fbMR1K4_Coating_States.stCoating2.stPMPS.sPmpsState := 'MR1K4:SOMS-B4C';
fbMR1K4_Coating_States.stCoating2.nEncoderCount := 5000141;

fbMR2K4_Coating_States.stCoating1.stPMPS.sPmpsState := 'MR2K4:KBO-SILICON';
fbMR2K4_Coating_States.stCoating1.nEncoderCount := 8701960;

fbMR2K4_Coating_States.stCoating2.stPMPS.sPmpsState := 'MR2K4:KBO-B4C';
fbMR2K4_Coating_States.stCoating2.nEncoderCount := 6636177;

fbMR3K4_Coating_States.stCoating1.stPMPS.sPmpsState := 'MR3K4:KBO-SILICON';
fbMR3K4_Coating_States.stCoating1.nEncoderCount := 4719890;

fbMR3K4_Coating_States.stCoating2.stPMPS.sPmpsState := 'MR3K4:KBO-B4C';
fbMR3K4_Coating_States.stCoating2.nEncoderCount := 8220029;

fbMR1K4_Coating_States(
    bEnable := TRUE,
    stMotionStage:=Main.M1,
    sCoating1Name:='Si',
    sCoating2Name:='B4C',
    fbArbiter:=GVL_PMPS.g_fbArbiter1,
    fbFFHWO:=GVL_PMPS.g_FastFaultOutput1,
    sPmpsDeviceName:='MR1K4:SOMS',
    sTransitionKey:= 'MR1K4:SOMS-TRANSITION');

// MR2K4 Coating States with PMPS
fbMR2K4_Coating_States(
    bEnable := TRUE,
    stMotionStage:=Main.M8,
    sCoating1Name:='Si',
    sCoating2Name:='B4C',
    fbArbiter:=GVL_PMPS.g_fbArbiter2,
    fbFFHWO:=GVL_PMPS.g_FastFaultOutput2,
    sPmpsDeviceName:='MR2K4:KBO',
    sTransitionKey:= 'MR2K4:KBO-TRANSITION'
);

// MR3K4 Coating States with PMPS
fbMR3K4_Coating_States(
    bEnable := TRUE,
    stMotionStage:=Main.M12,
    bVerticalCoating:=FALSE,
    sCoating1Name:='Si',
    sCoating2Name:='B4C',
    fbArbiter:=GVL_PMPS.g_fbArbiter2,
    fbFFHWO:=GVL_PMPS.g_FastFaultOutput2,
    sPmpsDeviceName:='MR3K4:KBO',
    sTransitionKey:= 'MR3K4:KBO-TRANSITION'
);

fbMR4K4XSetup(stPositionState:= fbMR4K4Default, bSetDefault :=TRUE);
fbMR4K4XSetup(stPositionState:=aMR4K4CoatingStatesX[ENUM_Si_B4C_Coating_States_1D.B4C],
    sName:='B4C',
    sPmpsState:='MR4K4:KBO-B4C',
    fDelta := 4.187,
    nEncoderCount:= 6727471
);
fbMR4K4XSetup(stPositionState:=aMR4K4CoatingStatesX[ENUM_Si_B4C_Coating_States_1D.Si],
    sName:='Si',
    sPmpsState:='MR4K4:KBO-SILICON',
    fDelta := 3.65,
    nEncoderCount:= 4322111
);
fbMR4K4_Coating_States(
    stMotionStage:=Main.M17,
    astPositionState:= aMR4K4CoatingStatesX,
    eEnumSet:= eMR4K4StateSet,
    eEnumGet:= eMR4K4StateGet,
    fbArbiter:=GVL_PMPS.g_fbArbiter2,
    fbFFHWO:=GVL_PMPS.g_FastFaultOutput3,
    bEnableMotion:=TRUE,
    bEnableBeamParams:=TRUE,
    sDeviceName:='MR4K4:KBO',
    sTransitionKey:= 'MR4K4:KBO-TRANSITION');

fbMR5K4YSetup(stPositionState:= fbMR5K4Default, bSetDefault :=TRUE);
fbMR5K4YSetup(stPositionState:=aMR5K4CoatingStatesY[ENUM_Si_B4C_Coating_States_1D.B4C],
    sName:='B4C',
    sPmpsState:='MR5K4:KBO-B4C',
    fDelta := 7.85,
    nEncoderCount:= 6785425
);
fbMR5K4YSetup(stPositionState:=aMR5K4CoatingStatesY[ENUM_Si_B4C_Coating_States_1D.Si],
    sName:='Si',
    sPmpsState:='MR5K4:KBO-SILICON',
    fDelta := 3.55,
    nEncoderCount:= 4265000
);
fbMR5K4_Coating_States(
    stMotionStage:=Main.M22,
    astPositionState:= aMR5K4CoatingStatesY,
    eEnumSet:= eMR5K4StateSet,
    eEnumGet:= eMR5K4StateGet,
    fbArbiter:=GVL_PMPS.g_fbArbiter2,
    fbFFHWO:=GVL_PMPS.g_FastFaultOutput3,
    bEnableMotion:=TRUE,
    bEnableBeamParams:=TRUE,
    sDeviceName:='MR5K4:KBO',
    sTransitionKey:= 'MR5K4:KBO-TRANSITION');

END_PROGRAM

// ---- POUs/PRG_PMPS.TcPOU
PROGRAM PRG_PMPS
VAR
    fb_vetoArbiter : FB_VetoArbiter;

    fbArbiterIO : FB_SubSysToArbiter_IO;

    ffFFO2ToFFO1 : FB_FastFault := (
        i_xAutoReset := TRUE,
        i_DevName := 'PMPS FFO2',
        i_Desc := 'Subordinate fast fault group, will clear on its own otherwise something is misconfigured in the diagnostic',
        i_TypeCode := 16#D);
//adding FFO3 for dream mirror so that we can veto dream mirror by ST4K4
   ffFFO3ToFFO1 : FB_FastFault := (
        i_xAutoReset := TRUE,
        i_DevName := 'PMPS FFO3',
        i_Desc := 'Subordinate fast fault group, will clear on its own otherwise something is misconfigured in the diagnostic',
        i_TypeCode := 16#D);

 //fbOutputStates : FB_StateParams;

    bMR1K1_IN : BOOL;
    bST3K4_IN : BOOL;
    bMR1K3_IN : BOOL;
    bST1K0_IN : BOOL;
    bST4K4_IN : BOOL;
END_VAR

MOTION_GVL.fbStandardPMPSDB(
    io_fbFFHWO:= GVL_PMPS.g_FastFaultOutput1,
    bEnable:=TRUE,
    sPLCName:='plc-tmo-optics'
);

P_StripeProtections();

bMR1K1_IN := PMPS.PMPS_GVL.stCurrentBeamParameters.aVetoDevices[PMPS.K_Stopper.MR1K1_IN]
            AND NOT PMPS.PMPS_GVL.stCurrentBeamParameters.aVetoDevices[PMPS.K_Stopper.MR1K1_OUT];

bST3K4_IN := PMPS.PMPS_GVL.stCurrentBeamParameters.aVetoDevices[PMPS.K_Stopper.ST3K4];
bST1K0_IN := PMPS.PMPS_GVL.stCurrentBeamParameters.aVetoDevices[PMPS.K_Stopper.ST1K0];

bMR1K3_IN := PMPS.PMPS_GVL.stCurrentBeamParameters.aVetodevices[PMPS.K_Stopper.MR1K3_IN]
    AND NOT PMPS.PMPS_GVL.stCurrentBeamParameters.aVetoDevices[PMPS.K_Stopper.MR1K3_OUT];

bST4K4_IN := PMPS.PMPS_GVL.stCurrentBeamParameters.aVetoDevices[PMPS.K_Stopper.ST4K4];

fbArbiterIO(i_bVeto:= bMR1K1_IN OR bMR1K3_IN, Arbiter := GVL_PMPS.g_fbArbiter1, fbFFHWO := GVL_PMPS.g_FastFaultOutput1);

ffFFO2ToFFO1(i_xOK := GVL_PMPS.g_FastFaultOutput2.q_xFastFaultOut, io_fbFFHWO := GVL_PMPS.g_FastFaultOutput1);
ffFFO3ToFFO1(i_xOK := GVL_PMPS.g_FastFaultOutput3.q_xFastFaultOut, io_fbFFHWO := GVL_PMPS.g_FastFaultOutput1);

GVL_PMPS.g_FastFaultOutput3.Execute(i_xVeto:= bMR1K1_IN OR bMR1K3_IN OR bST3K4_IN OR bST1K0_IN OR bST4K4_IN);

GVL_PMPS.g_FastFaultOutput2.Execute(i_xVeto:= bMR1K1_IN OR bMR1K3_IN OR bST3K4_IN OR bST1K0_IN);

GVL_PMPS.g_FastFaultOutput1.Execute(i_xVeto:= bMR1K1_IN OR bMR1K3_IN);

fb_vetoArbiter(bVeto := GVL_PMPS.g_FastFaultOutput2.i_xVeto, HigherAuthority := GVL_PMPS.g_fbArbiter1, LowerAuthority:= GVL_PMPS.g_fbArbiter2,
    FFO:= GVL_PMPS.g_FastFaultOutput1);

END_PROGRAM
